TEXTLIST TextList_tabvac_state
  0 = 'off'
  1 = 'idle'
  2 = 'waiting_vacuum_on'
  3 = 'waiting_vacuum_off'
  4 = 'on'
  5 = 'waiting_off'
  100 = 'error'
   = ''
END_TEXTLIST

(* stored: Version 1.1.0.1, ProductVersion 3.1.4024.11
   TextList TextList_tabvac_state: Id {dd174e8f-88ac-4f43-baab-10baf93d0e80} *)
